TYPE "BatchCheck_ShW"
VERSION : 0.1
   STRUCT
      Trigger : Bool;
      Q_ID : "batchID_ShW";
      IDResult : Int;
      IDResult1 : Array[1..10] of Int;
      Completed : Bool;
   END_STRUCT;

END_TYPE

